{attribute 'qualified_only'}
{attribute 'strict'}
TYPE Turntable :
(
	clockwise := 0,
	counterclockwise,
	switchoff
);
END_TYPE

(* stored: Version 1.1.0.1, ProductVersion 3.1.4022.12
   DUT Turntable: Id {6020a02d-be50-4094-9b44-6f47b259a55e} *)
